PROGRAM MAIN
VAR
	fbClockOneSecond : FB_CLOCK;
END_VAR

fbClockOneSecond(TIME_ON:=T#500MS, TIME_OFF:=T#500MS, OUT_CLK=>);

END_PROGRAM

(* stored: Version 1.1.0.1, ProductVersion 3.1.4024.12
   POU MAIN: Id {0f877463-314e-40d4-85f8-7b3707f59d66}, SpecialFunc None *)
